(* Logix 5000 project; controller HP_SSC01 vendor 1 type 14 code 67 rev 17.7; software revision 17.01; part 12 of 15 *)
(* tags used below, declared in another part *)
   A_C1_0200 : ALIAS FOR S_C1_FaultSafety.0;
   A_C1_0201 : ALIAS FOR S_C1_FaultSafety.1;
   A_C1_0202 : ALIAS FOR S_C1_FaultSafety.2;
   A_C1_0203 : ALIAS FOR S_C1_FaultSafety.3;
   A_C1_0204 : ALIAS FOR S_C1_FaultSafety.4;
   A_C1_0206 : ALIAS FOR S_C1_FaultSafety.6;
   A_C1_0208 : ALIAS FOR S_C1_FaultSafety.8;
   A_C1_0209 : ALIAS FOR S_C1_FaultSafety.9;
   A_C1_0210 : ALIAS FOR S_C1_FaultSafety.10;
   A_C1_0211 : ALIAS FOR S_C1_FaultSafety.11;
   A_C1_0216 : ALIAS FOR S_C1_FaultSafety.16;
   A_C1_0217 : ALIAS FOR S_C1_FaultSafety.17;
   A_C1_0218 : ALIAS FOR S_C1_FaultSafety.18;
   A_C1_0219 : ALIAS FOR S_C1_FaultSafety.19;
   A_C1_0220 : ALIAS FOR S_C1_FaultSafety.20;
   A_C1_0221 : ALIAS FOR S_C1_FaultSafety.21;
   A_C1_0222 : ALIAS FOR S_C1_FaultSafety.22;
   A_C1_0223 : ALIAS FOR S_C1_FaultSafety.23;
   A_C1_0224 : ALIAS FOR S_C1_FaultSafety.24;
   A_C1_0230 : ALIAS FOR S_C1_FaultSafety.30;
   A_C1_0231 : ALIAS FOR S_C1_FaultSafety.31;
   A_C2_0200 : ALIAS FOR S_C2_FaultSafety.0;
   A_C2_0201 : ALIAS FOR S_C2_FaultSafety.1;
   A_C2_0210 : ALIAS FOR S_C2_FaultSafety.10;
   A_C2_0211 : ALIAS FOR S_C2_FaultSafety.11;
   A_C3_0200 : ALIAS FOR S_C3_FaultSafety.0;
   A_C3_0201 : ALIAS FOR S_C3_FaultSafety.1;
   A_C3_0210 : ALIAS FOR S_C3_FaultSafety.10;
   A_C3_0211 : ALIAS FOR S_C3_FaultSafety.11;
   A_S01_0103 : ALIAS FOR System_FaultSafeIO.3;
   A_S01_0104 : ALIAS FOR System_FaultSafeIO.4;
   A_S01_0105 : ALIAS FOR System_FaultSafeIO.5;
   A_S01_0116 : ALIAS FOR System_FaultSafeIO.16;
   A_S01_0117 : ALIAS FOR System_FaultSafeIO.17;
   A_S01_0118 : ALIAS FOR System_FaultSafeIO.18;
   A_S01_0119 : ALIAS FOR System_FaultSafeIO.19;
   A_S01_0120 : ALIAS FOR System_FaultSafeIO.20;
   A_S01_0122 : ALIAS FOR System_FaultSafeIO.22;
   A_S01_0123 : ALIAS FOR System_FaultSafeIO.23;
   A_S01_0124 : ALIAS FOR System_FaultSafeIO.24;
   A_S01_0201 : ALIAS FOR System_FaultSafety.1;
   A_S01_0204 : ALIAS FOR System_FaultSafety.4;
   A_S01_0206 : ALIAS FOR System_FaultSafety.6;
   A_S01_0208 : ALIAS FOR System_FaultSafety.8;
   A_S01_0209 : ALIAS FOR System_FaultSafety.9;
   A_S01_0210 : ALIAS FOR System_FaultSafety.10;
   A_S01_0211 : ALIAS FOR System_FaultSafety.11;
   A_S01_0212 : ALIAS FOR System_FaultSafety.12;
   A_S01_0213 : ALIAS FOR System_FaultSafety.13;
   A_S01_0216 : ALIAS FOR System_FaultSafety.16;
   C01_SafeMemory : Udt_Carsl_SafeData;
   ONS_STFault : DINT;
   Rail_Bypass1 : ALIAS FOR SSC01_Safe1:I.Pt06Data;
   Rail_Bypass2 : ALIAS FOR SSC01_Safe1:I.Pt07Data;
   RAIL_ENABLE_LH1 : ALIAS FOR SSC01_Safe1:I.Pt00Data;
   RAIL_ENABLE_LH2 : ALIAS FOR SSC01_Safe1:I.Pt01Data;
   RAIL_ENABLE_LH3 : ALIAS FOR SSC01_Safe1:I.Pt02Data;
   RAIL_ENABLE_RH1 : ALIAS FOR SSC01_Safe1:I.Pt03Data;
   RAIL_ENABLE_RH2 : ALIAS FOR SSC01_Safe1:I.Pt04Data;
   RAIL_ENABLE_RH3 : ALIAS FOR SSC01_Safe1:I.Pt05Data;
   RAIL_SHUNT_FDBK_LH1 : ALIAS FOR SSC01_Safe3:I.Pt00Data;
   RAIL_SHUNT_FDBK_LH2 : ALIAS FOR SSC01_Safe3:I.Pt01Data;
   RAIL_SHUNT_FDBK_LH3 : ALIAS FOR SSC01_Safe3:I.Pt02Data;
   Rail_Shunt_Fdbk_OK : BOOL;
   RAIL_SHUNT_FDBK_RH1 : ALIAS FOR SSC01_Safe3:I.Pt03Data;
   RAIL_SHUNT_FDBK_RH2 : ALIAS FOR SSC01_Safe3:I.Pt04Data;
   RAIL_SHUNT_FDBK_RH3 : ALIAS FOR SSC01_Safe3:I.Pt05Data;
   RAIL_SHUNT_LH1 : ALIAS FOR SSC01_Safe1:O.Pt00Data;
   RAIL_SHUNT_LH2 : ALIAS FOR SSC01_Safe1:O.Pt01Data;
   RAIL_SHUNT_LH3 : ALIAS FOR SSC01_Safe1:O.Pt02Data;
   RAIL_SHUNT_RH1 : ALIAS FOR SSC01_Safe1:O.Pt03Data;
   RAIL_SHUNT_RH2 : ALIAS FOR SSC01_Safe1:O.Pt04Data;
   RAIL_SHUNT_RH3 : ALIAS FOR SSC01_Safe1:O.Pt05Data;
   RCS_CMD_EvacToStation : BOOL;
   RCS_CMD_GoNearOnPath : BOOL;
   RCS_Cmd_Mismatch_TON : TIMER;
   RCS_CMD_RunInAuto : BOOL;
   RCS_Cmd_Unknown : BOOL;
   RCS_MasterClock : ALIAS FOR RCS_SafeMemory_S01.Master_Clock;
   RCS_MasterPositionMOD7000 : DINT;
   RCS_MasterPositionMOD7000X1000 : DINT;
   RCS_PwrDisc_RIN : REDUNDANT_INPUT;
   RCS_SafeMemory_S01 : Udt_RCS_SafeData;
   RCS_SyncMotionEnable : BOOL;
   S_C01_MStopOK : BOOL;
   S_C02_MStopOK : BOOL;
   S_C03_MStopOK : BOOL;
   S_C1_AtEvacSpeed : BOOL;
   S_C1_BrakeRelease : ALIAS FOR C1_Safe:O.Pt06Data;
   S_C1_BrakeReleaseSelected : BOOL;
   S_C1_BrakeTest : BOOL;
   S_C1_CircuitReset : BOOL;
   S_C1_DrawbridgeInputOK : BOOL;
   S_C1_DrawbridgeRIN : REDUNDANT_INPUT;
   S_C1_DumpValveRelease : ALIAS FOR C1_Safe:O.Pt05Data;
   S_C1_DumpValveReleaseSelected : BOOL;
   S_C1_EncoderBuffer : DINT[4];
   S_C1_EncoderChange : DINT;
   S_C1_EncoderCounter : DINT;
   S_C1_EncoderCounts : DINT;
   S_C1_EncoderPositionAtHome : DINT;
   S_C1_EncoderPositionAtHomeSet : BOOL;
   S_C1_EncoderPositionDegree : DINT;
   S_C1_EncoderRev : DINT;
   S_C1_EncoderRevX1000 : DINT;
   S_C1_EncoderTemp : DINT;
   S_C1_EncoderTemp2 : DINT;
   S_C1_EvacOk : BOOL;
   S_C1_ExecuteInputOK : BOOL;
   S_C1_FaultReset : BOOL;
   S_C1_FaultSafety : DINT;
   S_C1_FaultSafety_OK : BOOL;
   S_C1_FaultStandard_OK : BOOL;
   S_C1_FaultTimer : TIMER[8];
   S_C1_Homed : BOOL;
   S_C1_HomeInputStatus : BOOL;
   S_C1_HomeSafePE : ALIAS FOR C1_Safe:I.Pt04Data;
   S_C1_InEvacPosition : BOOL;
   S_C1_ModeLocal : BOOL;
   S_C1_ModeRemote : BOOL;
   S_C1_MotorActualPositionX1000 : DINT;
   S_C1_MotorAverageVelocityX1000 : DINT;
   S_C1_MotorToEncoderError : DINT;
   S_C1_MStop : EMERGENCY_STOP;
   S_C1_MSTOP_InputOK : BOOL;
   S_C1_OffPath : BOOL;
   S_C1_OnPath : BOOL;
   S_C1_ONS_Fault : BOOL;
   S_C1_OutputEnable : BOOL;
   S_C1_PressureOK : ALIAS FOR C1_Safe:I.Pt05Data;
   S_C1_RemoteBrakeAndHomeSequence : DINT;
   S_C1_ReverseMotionDebounce : TIMER;
   S_C1_SAFE_OFF_FDBK1 : ALIAS FOR C1_Safe:I.Pt01Data;
   S_C1_SAFE_OFF_FDBK2 : ALIAS FOR C1_Safe:I.Pt00Data;
   S_C1_SafeOff_ROUT : REDUNDANT_OUTPUT;
   S_C1_SafeOffInputOK : BOOL;
   S_C1_SetEncoderHomePosition : BOOL;
   S_C1_Stop0 : BOOL;
   S_C1_Stop0_OK : BOOL;
   S_C1_Stop1 : BOOL;
   S_C1_Stop1_OK : BOOL;
   S_C2_EvacOK : BOOL;
   S_C2_ModeLocal : BOOL;
   S_C2_ModeRemote : BOOL;
   S_C2_OffPath : BOOL;
   S_C2_OnPath : BOOL;
   S_C2_Stop0 : BOOL;
   S_C2_Stop0_OK : BOOL;
   S_C2_Stop1 : BOOL;
   S_C2_Stop1_OK : BOOL;
   S_C3_EvacOK : BOOL;
   S_C3_ModeLocal : BOOL;
   S_C3_ModeRemote : BOOL;
   S_C3_OffPath : BOOL;
   S_C3_OnPath : BOOL;
   S_C3_Stop0 : BOOL;
   S_C3_Stop0_OK : BOOL;
   S_C3_Stop1 : BOOL;
   S_C3_Stop1_OK : BOOL;
   S_DeviceNet_OK : BOOL;
   S_EncoderRollover : DINT;
   S_EvacToStationTON : TIMER;
   S_FaultReset : BOOL;
   S_RCS_EvacSpeedStart_TON : TIMER;
   S_RCS_MasterPositionDegrees : DINT;
   S_S01_Mode_Remote : BOOL;
   S_S01_NearOnPath : BOOL;
   S_S01_OnPath : BOOL;
   S_S01_Ready : BOOL;
   S_System_FaultStandard : DINT;
   SSC_Auto_Decel1 : BOOL;
   SSC_Mode_Local_LT : ALIAS FOR SSC01_Safe3:O.Pt00Data;
   SSC_Mode_Remote_LT : ALIAS FOR SSC01_Safe3:O.Pt02Data;
   SSC_NoStopFault : BOOL;
   SSC_Rail_BypassOK : BOOL;
   SSC_Rail_InputsOK : BOOL;
   SSC_RailShuntOK : BOOL;
   SSC_Ready_LT : ALIAS FOR SSC01_Safe3:O.Pt01Data;
   SSC_SafeFlt_OK : BOOL;
   SSC_SafetyIO_OK : BOOL;
   SSC_StdFlt_OK : BOOL;
   SSC_Stop0_OK : BOOL;
   SSC_Stop1_OK : BOOL;
   ST_NoScan_Comment : BOOL;
   STS_Rail_Bypass_InputOK : BOOL;
   STS_RCS_PwrDisc_InputOK : BOOL;
   STS_Status_OK : BOOL;
   System_FaultSafeIO : DINT;
   System_FaultSafety : DINT;
   Tmr_Rail_Shunt : TIMER[7];
(* Safe_SSC, continued *)

ROUTINE ST10_PositionHandling   (* ladder *)
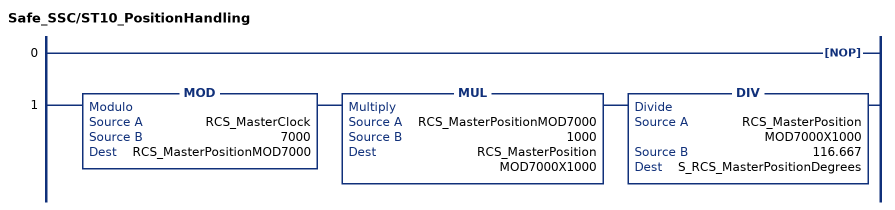
   0: NOP();
   1: MOD(RCS_MasterClock,7000,RCS_MasterPositionMOD7000)MUL(RCS_MasterPositionMOD7000,1000,RCS_MasterPositionMOD7000X1000)DIV(RCS_MasterPositionMOD7000X1000,116.667,S_RCS_MasterPositionDegrees);
END_ROUTINE

ROUTINE ST21_RailShunt   (* ladder *)
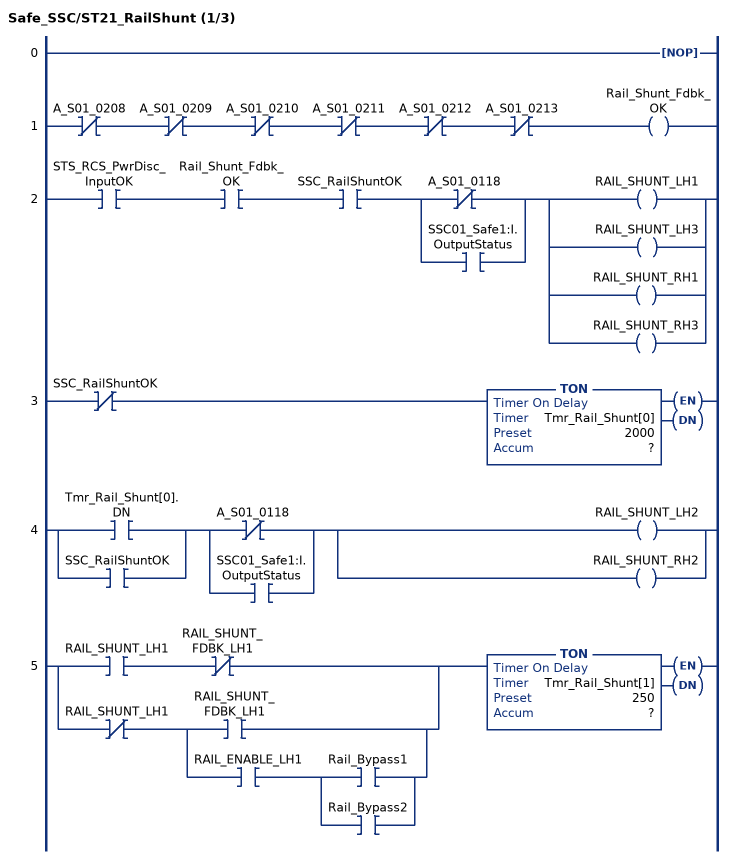
   0: NOP();
   1: XIO(A_S01_0208)XIO(A_S01_0209)XIO(A_S01_0210)XIO(A_S01_0211)XIO(A_S01_0212)XIO(A_S01_0213)OTE(Rail_Shunt_Fdbk_OK);
   2: XIC(STS_RCS_PwrDisc_InputOK)XIC(Rail_Shunt_Fdbk_OK)XIC(SSC_RailShuntOK)[XIO(A_S01_0118) ,XIC(SSC01_Safe1:I.OutputStatus) ][OTE(RAIL_SHUNT_LH1) ,OTE(RAIL_SHUNT_LH3) ,OTE(RAIL_SHUNT_RH1) ,OTE(RAIL_SHUNT_RH3) ];
   3: XIO(SSC_RailShuntOK)TON(Tmr_Rail_Shunt[0],?,?);
   4: [XIC(Tmr_Rail_Shunt[0].DN) ,XIC(SSC_RailShuntOK) ][XIO(A_S01_0118) ,XIC(SSC01_Safe1:I.OutputStatus) ][OTE(RAIL_SHUNT_LH2) ,OTE(RAIL_SHUNT_RH2) ];
   5: [XIC(RAIL_SHUNT_LH1) XIO(RAIL_SHUNT_FDBK_LH1) ,XIO(RAIL_SHUNT_LH1) [XIC(RAIL_SHUNT_FDBK_LH1) ,XIC(RAIL_ENABLE_LH1) [XIC(Rail_Bypass1) ,XIC(Rail_Bypass2) ] ] ]TON(Tmr_Rail_Shunt[1],?,?);
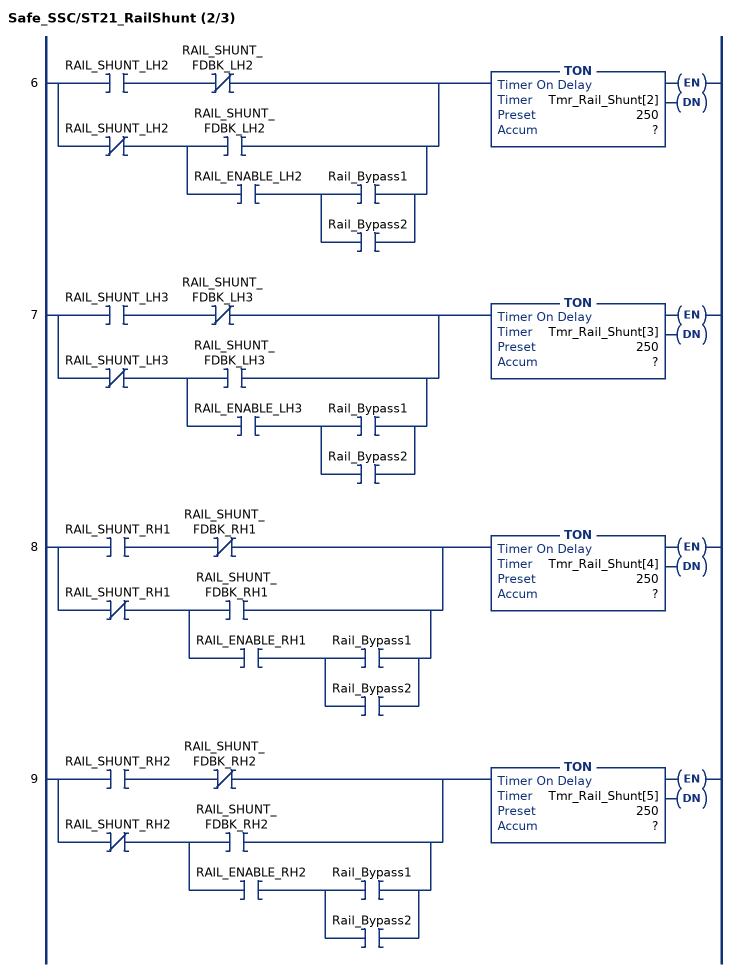
   6: [XIC(RAIL_SHUNT_LH2) XIO(RAIL_SHUNT_FDBK_LH2) ,XIO(RAIL_SHUNT_LH2) [XIC(RAIL_SHUNT_FDBK_LH2) ,XIC(RAIL_ENABLE_LH2) [XIC(Rail_Bypass1) ,XIC(Rail_Bypass2) ] ] ]TON(Tmr_Rail_Shunt[2],?,?);
   7: [XIC(RAIL_SHUNT_LH3) XIO(RAIL_SHUNT_FDBK_LH3) ,XIO(RAIL_SHUNT_LH3) [XIC(RAIL_SHUNT_FDBK_LH3) ,XIC(RAIL_ENABLE_LH3) [XIC(Rail_Bypass1) ,XIC(Rail_Bypass2) ] ] ]TON(Tmr_Rail_Shunt[3],?,?);
   8: [XIC(RAIL_SHUNT_RH1) XIO(RAIL_SHUNT_FDBK_RH1) ,XIO(RAIL_SHUNT_RH1) [XIC(RAIL_SHUNT_FDBK_RH1) ,XIC(RAIL_ENABLE_RH1) [XIC(Rail_Bypass1) ,XIC(Rail_Bypass2) ] ] ]TON(Tmr_Rail_Shunt[4],?,?);
   9: [XIC(RAIL_SHUNT_RH2) XIO(RAIL_SHUNT_FDBK_RH2) ,XIO(RAIL_SHUNT_RH2) [XIC(RAIL_SHUNT_FDBK_RH2) ,XIC(RAIL_ENABLE_RH2) [XIC(Rail_Bypass1) ,XIC(Rail_Bypass2) ] ] ]TON(Tmr_Rail_Shunt[5],?,?);
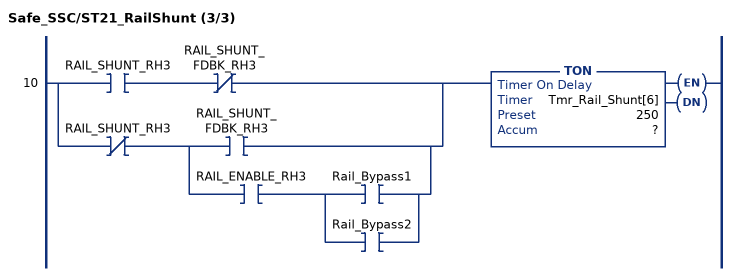
   10: [XIC(RAIL_SHUNT_RH3) XIO(RAIL_SHUNT_FDBK_RH3) ,XIO(RAIL_SHUNT_RH3) [XIC(RAIL_SHUNT_FDBK_RH3) ,XIC(RAIL_ENABLE_RH3) [XIC(Rail_Bypass1) ,XIC(Rail_Bypass2) ] ] ]TON(Tmr_Rail_Shunt[6],?,?);
END_ROUTINE

ROUTINE ST23_GenOutputs   (* ladder *)
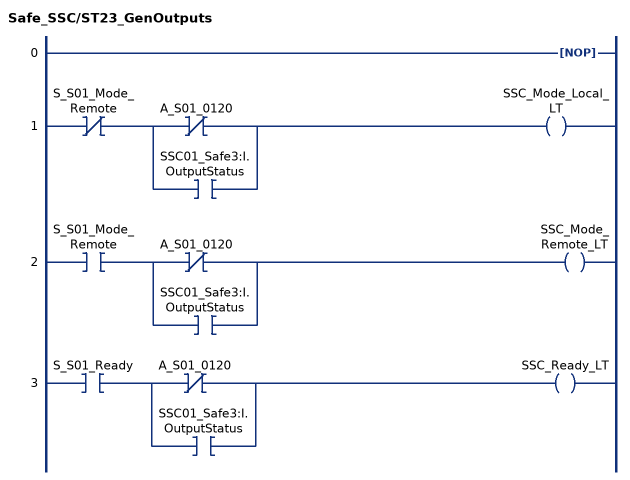
   0: NOP();
   1: XIO(S_S01_Mode_Remote)[XIO(A_S01_0120) ,XIC(SSC01_Safe3:I.OutputStatus) ]OTE(SSC_Mode_Local_LT);
   2: XIC(S_S01_Mode_Remote)[XIO(A_S01_0120) ,XIC(SSC01_Safe3:I.OutputStatus) ]OTE(SSC_Mode_Remote_LT);
   3: XIC(S_S01_Ready)[XIO(A_S01_0120) ,XIC(SSC01_Safe3:I.OutputStatus) ]OTE(SSC_Ready_LT);
END_ROUTINE

ROUTINE ST90_Faults   (* ladder *)
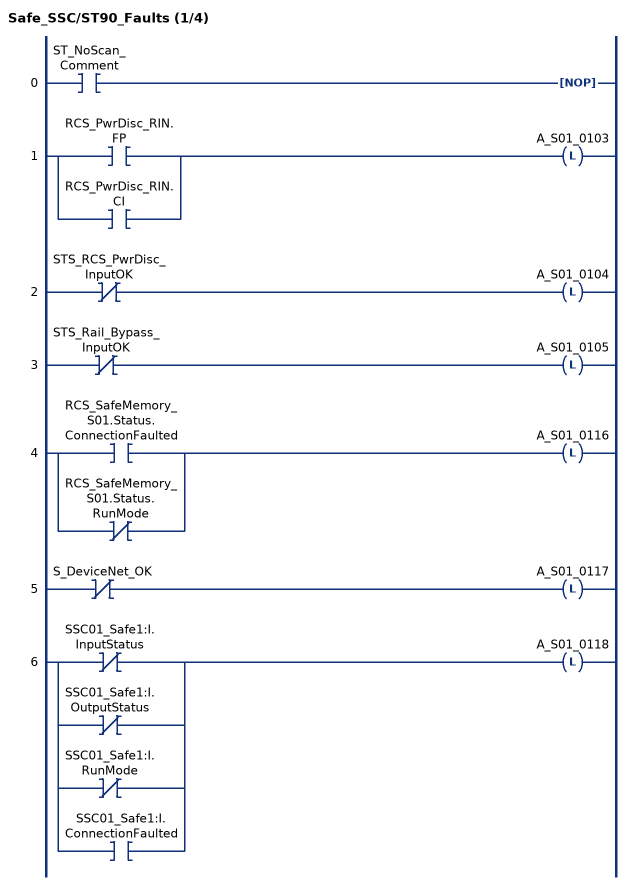
   0: XIC(ST_NoScan_Comment)NOP();
   1: [XIC(RCS_PwrDisc_RIN.FP) ,XIC(RCS_PwrDisc_RIN.CI) ]OTL(A_S01_0103);
   2: XIO(STS_RCS_PwrDisc_InputOK)OTL(A_S01_0104);
   3: XIO(STS_Rail_Bypass_InputOK)OTL(A_S01_0105);
   4: [XIC(RCS_SafeMemory_S01.Status.ConnectionFaulted) ,XIO(RCS_SafeMemory_S01.Status.RunMode) ]OTL(A_S01_0116);
   5: XIO(S_DeviceNet_OK)OTL(A_S01_0117);
   6: [XIO(SSC01_Safe1:I.InputStatus) ,XIO(SSC01_Safe1:I.OutputStatus) ,XIO(SSC01_Safe1:I.RunMode) ,XIC(SSC01_Safe1:I.ConnectionFaulted) ]OTL(A_S01_0118);
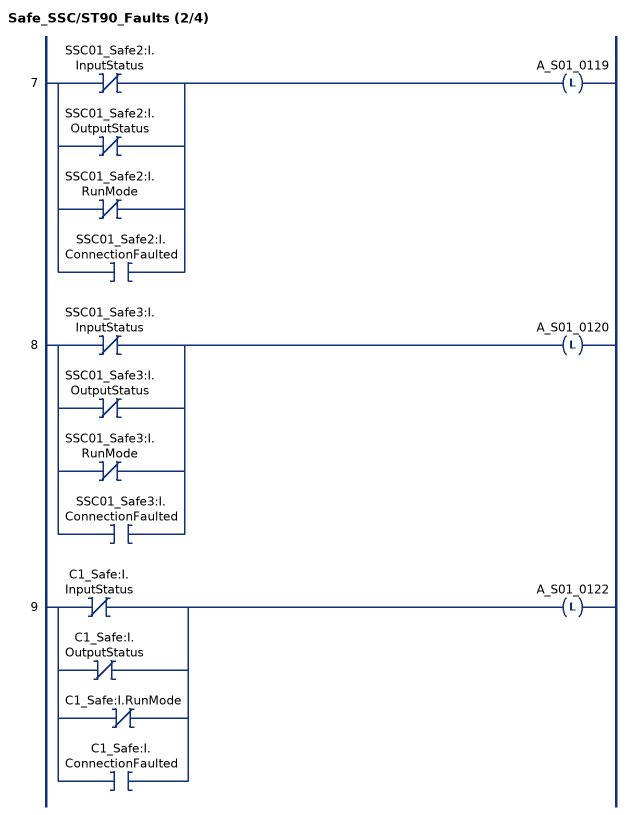
   7: [XIO(SSC01_Safe2:I.InputStatus) ,XIO(SSC01_Safe2:I.OutputStatus) ,XIO(SSC01_Safe2:I.RunMode) ,XIC(SSC01_Safe2:I.ConnectionFaulted) ]OTL(A_S01_0119);
   8: [XIO(SSC01_Safe3:I.InputStatus) ,XIO(SSC01_Safe3:I.OutputStatus) ,XIO(SSC01_Safe3:I.RunMode) ,XIC(SSC01_Safe3:I.ConnectionFaulted) ]OTL(A_S01_0120);
   9: [XIO(C1_Safe:I.InputStatus) ,XIO(C1_Safe:I.OutputStatus) ,XIO(C1_Safe:I.RunMode) ,XIC(C1_Safe:I.ConnectionFaulted) ]OTL(A_S01_0122);
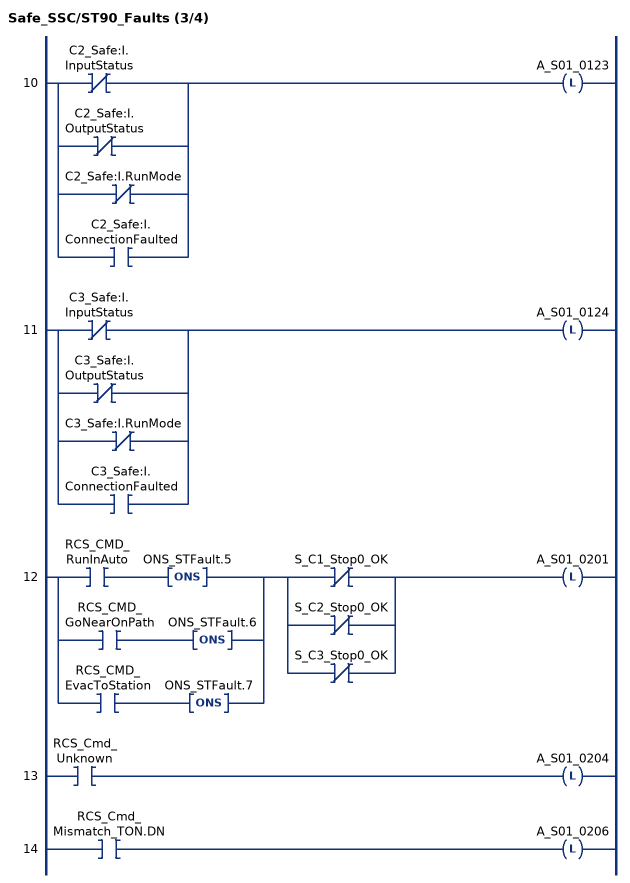
   10: [XIO(C2_Safe:I.InputStatus) ,XIO(C2_Safe:I.OutputStatus) ,XIO(C2_Safe:I.RunMode) ,XIC(C2_Safe:I.ConnectionFaulted) ]OTL(A_S01_0123);
   11: [XIO(C3_Safe:I.InputStatus) ,XIO(C3_Safe:I.OutputStatus) ,XIO(C3_Safe:I.RunMode) ,XIC(C3_Safe:I.ConnectionFaulted) ]OTL(A_S01_0124);
   12: [XIC(RCS_CMD_RunInAuto) ONS(ONS_STFault.5) ,XIC(RCS_CMD_GoNearOnPath) ONS(ONS_STFault.6) ,XIC(RCS_CMD_EvacToStation) ONS(ONS_STFault.7) ][XIO(S_C1_Stop0_OK) ,XIO(S_C2_Stop0_OK) ,XIO(S_C3_Stop0_OK) ]OTL(A_S01_0201);
   13: XIC(RCS_Cmd_Unknown)OTL(A_S01_0204);
   14: XIC(RCS_Cmd_Mismatch_TON.DN)OTL(A_S01_0206);
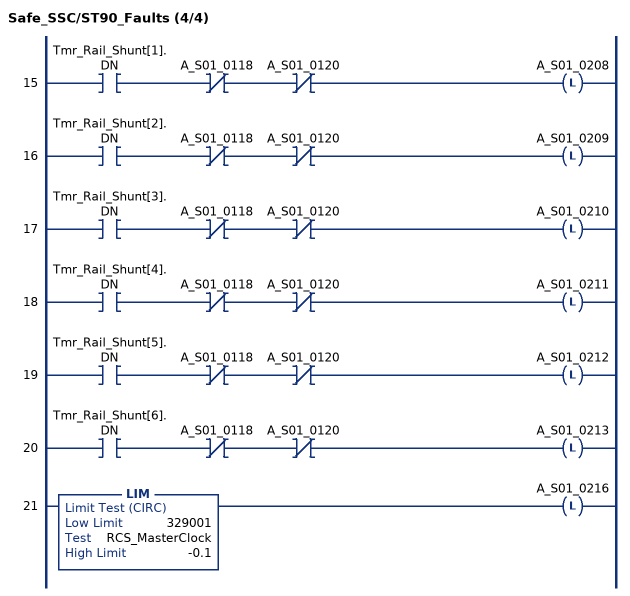
   15: XIC(Tmr_Rail_Shunt[1].DN)XIO(A_S01_0118)XIO(A_S01_0120)OTL(A_S01_0208);
   16: XIC(Tmr_Rail_Shunt[2].DN)XIO(A_S01_0118)XIO(A_S01_0120)OTL(A_S01_0209);
   17: XIC(Tmr_Rail_Shunt[3].DN)XIO(A_S01_0118)XIO(A_S01_0120)OTL(A_S01_0210);
   18: XIC(Tmr_Rail_Shunt[4].DN)XIO(A_S01_0118)XIO(A_S01_0120)OTL(A_S01_0211);
   19: XIC(Tmr_Rail_Shunt[5].DN)XIO(A_S01_0118)XIO(A_S01_0120)OTL(A_S01_0212);
   20: XIC(Tmr_Rail_Shunt[6].DN)XIO(A_S01_0118)XIO(A_S01_0120)OTL(A_S01_0213);
   21: LIM(329001,RCS_MasterClock,-0.1)OTL(A_S01_0216);
END_ROUTINE

ROUTINE ST91_FaultList   (* ladder *)
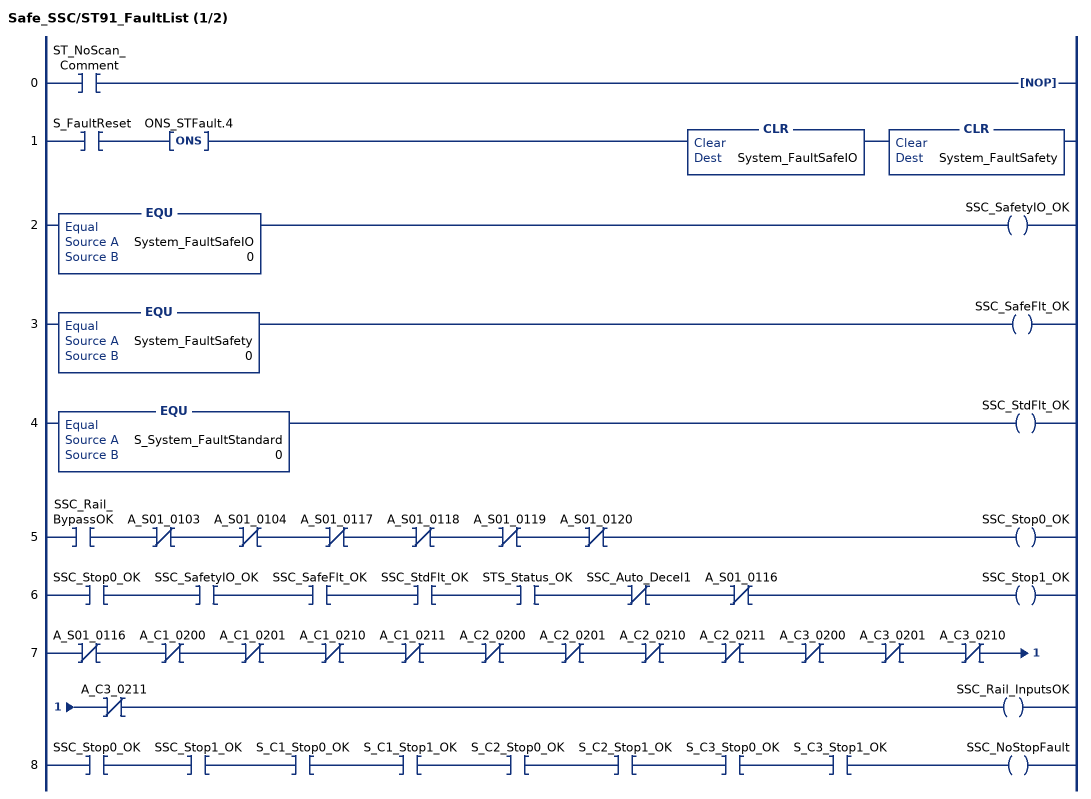
   0: XIC(ST_NoScan_Comment)NOP();
   1: XIC(S_FaultReset)ONS(ONS_STFault.4)CLR(System_FaultSafeIO)CLR(System_FaultSafety);
   2: EQU(System_FaultSafeIO,0)OTE(SSC_SafetyIO_OK);
   3: EQU(System_FaultSafety,0)OTE(SSC_SafeFlt_OK);
   4: EQU(S_System_FaultStandard,0)OTE(SSC_StdFlt_OK);
   5: XIC(SSC_Rail_BypassOK)XIO(A_S01_0103)XIO(A_S01_0104)XIO(A_S01_0117)XIO(A_S01_0118)XIO(A_S01_0119)XIO(A_S01_0120)OTE(SSC_Stop0_OK);
   6: XIC(SSC_Stop0_OK)XIC(SSC_SafetyIO_OK)XIC(SSC_SafeFlt_OK)XIC(SSC_StdFlt_OK)XIC(STS_Status_OK)XIO(SSC_Auto_Decel1)XIO(A_S01_0116)OTE(SSC_Stop1_OK);
   7: XIO(A_S01_0116)XIO(A_C1_0200)XIO(A_C1_0201)XIO(A_C1_0210)XIO(A_C1_0211)XIO(A_C2_0200)XIO(A_C2_0201)XIO(A_C2_0210)XIO(A_C2_0211)XIO(A_C3_0200)XIO(A_C3_0201)XIO(A_C3_0210)XIO(A_C3_0211)OTE(SSC_Rail_InputsOK);
   8: XIC(SSC_Stop0_OK)XIC(SSC_Stop1_OK)XIC(S_C1_Stop0_OK)XIC(S_C1_Stop1_OK)XIC(S_C2_Stop0_OK)XIC(S_C2_Stop1_OK)XIC(S_C3_Stop0_OK)XIC(S_C3_Stop1_OK)OTE(SSC_NoStopFault);
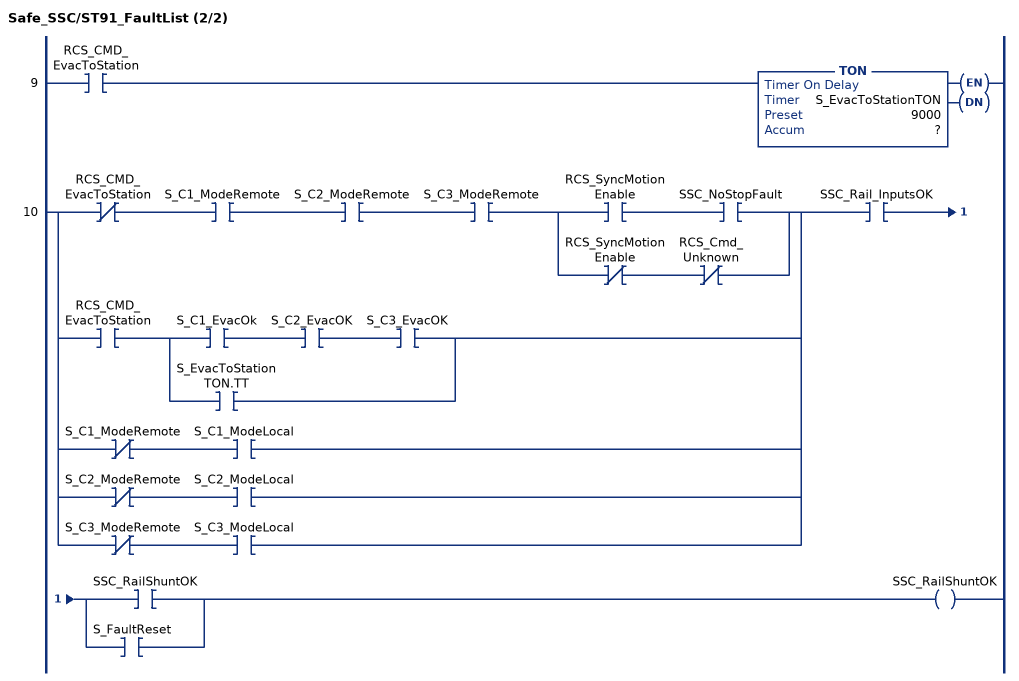
   9: XIC(RCS_CMD_EvacToStation)TON(S_EvacToStationTON,?,?);
   10: [XIO(RCS_CMD_EvacToStation) XIC(S_C1_ModeRemote) XIC(S_C2_ModeRemote) XIC(S_C3_ModeRemote) [XIC(RCS_SyncMotionEnable) XIC(SSC_NoStopFault) ,XIO(RCS_SyncMotionEnable) XIO(RCS_Cmd_Unknown) ] ,XIC(RCS_CMD_EvacToStation) [XIC(S_C1_EvacOk) XIC(S_C2_EvacOK) XIC(S_C3_EvacOK) ,XIC(S_EvacToStationTON.TT) ] ,XIO(S_C1_ModeRemote) XIC(S_C1_ModeLocal) ,XIO(S_C2_ModeRemote) XIC(S_C2_ModeLocal) ,XIO(S_C3_ModeRemote) XIC(S_C3_ModeLocal) ]XIC(SSC_Rail_InputsOK)[XIC(SSC_RailShuntOK) ,XIC(S_FaultReset) ]OTE(SSC_RailShuntOK);
END_ROUTINE

ROUTINE ST99_CommToRCS   (* ladder *)
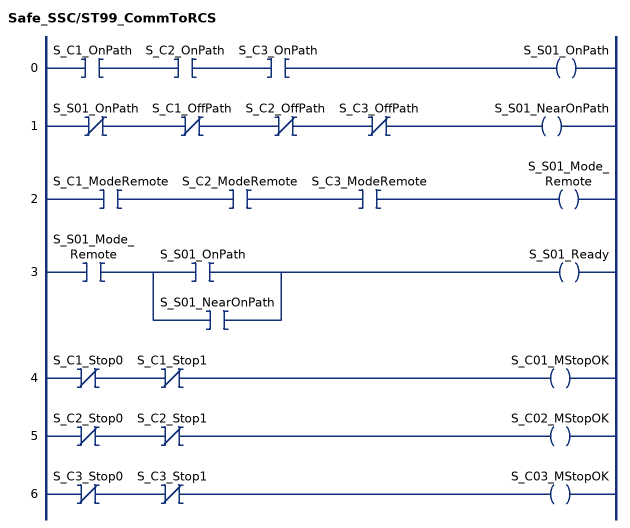
   0: XIC(S_C1_OnPath)XIC(S_C2_OnPath)XIC(S_C3_OnPath)OTE(S_S01_OnPath);
   1: XIO(S_S01_OnPath)XIO(S_C1_OffPath)XIO(S_C2_OffPath)XIO(S_C3_OffPath)OTE(S_S01_NearOnPath);
   2: XIC(S_C1_ModeRemote)XIC(S_C2_ModeRemote)XIC(S_C3_ModeRemote)OTE(S_S01_Mode_Remote);
   3: XIC(S_S01_Mode_Remote)[XIC(S_S01_OnPath) ,XIC(S_S01_NearOnPath) ]OTE(S_S01_Ready);
   4: XIO(S_C1_Stop0)XIO(S_C1_Stop1)OTE(S_C01_MStopOK);
   5: XIO(S_C2_Stop0)XIO(S_C2_Stop1)OTE(S_C02_MStopOK);
   6: XIO(S_C3_Stop0)XIO(S_C3_Stop1)OTE(S_C03_MStopOK);
END_ROUTINE
END_PROGRAM

PROGRAM SafeCarousel1   (* main routine SC100_Main *)

ROUTINE SC100_Main   (* ladder *)
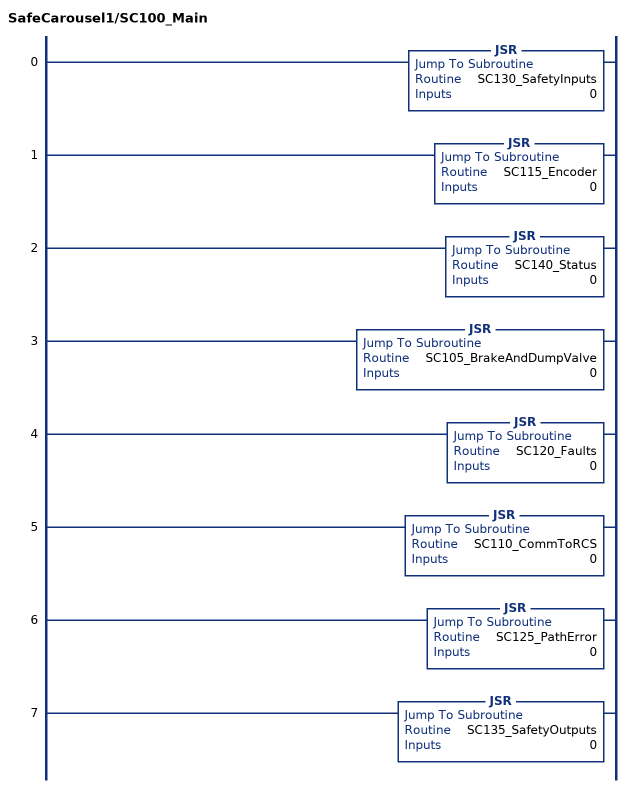
   0: JSR(SC130_SafetyInputs,0);
   1: JSR(SC115_Encoder,0);
   2: JSR(SC140_Status,0);
   3: JSR(SC105_BrakeAndDumpValve,0);
   4: JSR(SC120_Faults,0);
   5: JSR(SC110_CommToRCS,0);
   6: JSR(SC125_PathError,0);
   7: JSR(SC135_SafetyOutputs,0);
END_ROUTINE

ROUTINE SC105_BrakeAndDumpValve   (* ladder *)
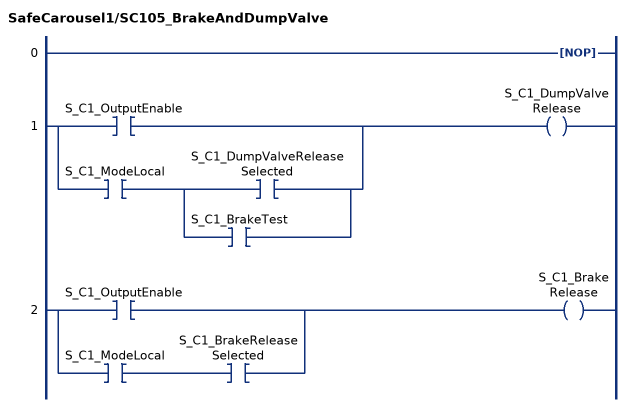
   0: NOP();
   1: [XIC(S_C1_OutputEnable) ,XIC(S_C1_ModeLocal) [XIC(S_C1_DumpValveReleaseSelected) ,XIC(S_C1_BrakeTest) ] ]OTE(S_C1_DumpValveRelease);
   2: [XIC(S_C1_OutputEnable) ,XIC(S_C1_ModeLocal) XIC(S_C1_BrakeReleaseSelected) ]OTE(S_C1_BrakeRelease);
END_ROUTINE

ROUTINE SC110_CommToRCS   (* ladder *)
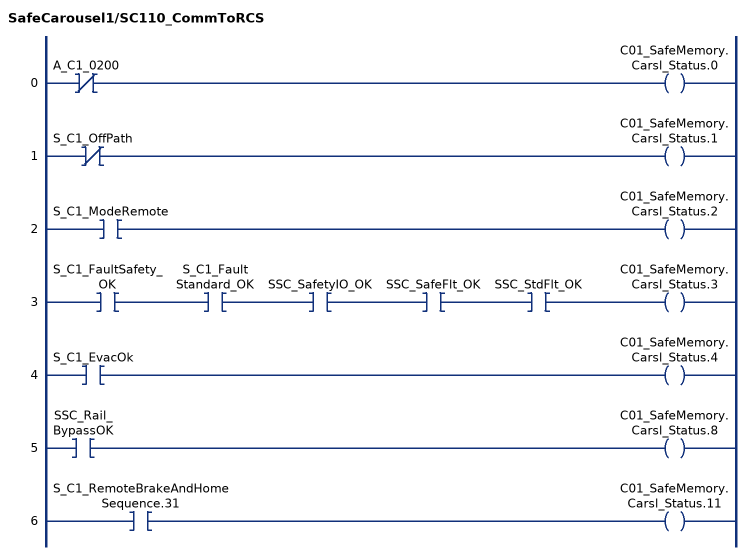
   0: XIO(A_C1_0200)OTE(C01_SafeMemory.Carsl_Status.0);
   1: XIO(S_C1_OffPath)OTE(C01_SafeMemory.Carsl_Status.1);
   2: XIC(S_C1_ModeRemote)OTE(C01_SafeMemory.Carsl_Status.2);
   3: XIC(S_C1_FaultSafety_OK)XIC(S_C1_FaultStandard_OK)XIC(SSC_SafetyIO_OK)XIC(SSC_SafeFlt_OK)XIC(SSC_StdFlt_OK)OTE(C01_SafeMemory.Carsl_Status.3);
   4: XIC(S_C1_EvacOk)OTE(C01_SafeMemory.Carsl_Status.4);
   5: XIC(SSC_Rail_BypassOK)OTE(C01_SafeMemory.Carsl_Status.8);
   6: XIC(S_C1_RemoteBrakeAndHomeSequence.31)OTE(C01_SafeMemory.Carsl_Status.11);
END_ROUTINE

ROUTINE SC115_Encoder   (* ladder *)
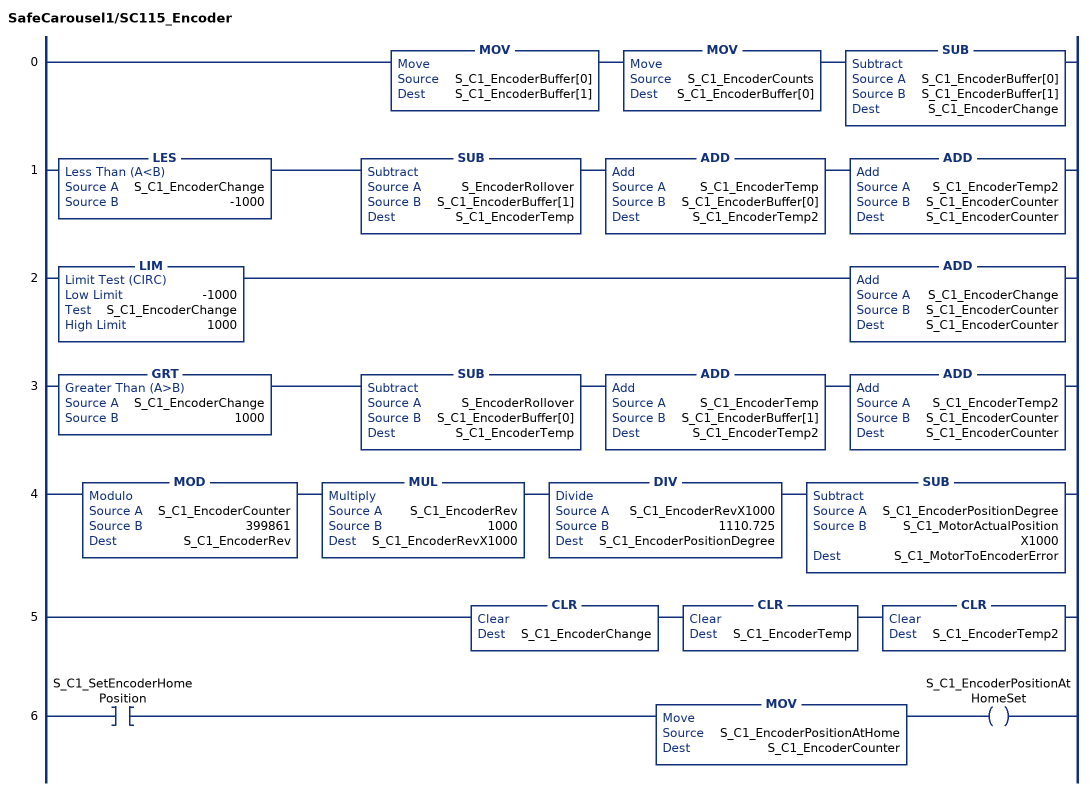
   0: MOV(S_C1_EncoderBuffer[0],S_C1_EncoderBuffer[1])MOV(S_C1_EncoderCounts,S_C1_EncoderBuffer[0])SUB(S_C1_EncoderBuffer[0],S_C1_EncoderBuffer[1],S_C1_EncoderChange);
   1: LES(S_C1_EncoderChange,-1000)SUB(S_EncoderRollover,S_C1_EncoderBuffer[1],S_C1_EncoderTemp)ADD(S_C1_EncoderTemp,S_C1_EncoderBuffer[0],S_C1_EncoderTemp2)ADD(S_C1_EncoderTemp2,S_C1_EncoderCounter,S_C1_EncoderCounter);
   2: LIM(-1000,S_C1_EncoderChange,1000)ADD(S_C1_EncoderChange,S_C1_EncoderCounter,S_C1_EncoderCounter);
   3: GRT(S_C1_EncoderChange,1000)SUB(S_EncoderRollover,S_C1_EncoderBuffer[0],S_C1_EncoderTemp)ADD(S_C1_EncoderTemp,S_C1_EncoderBuffer[1],S_C1_EncoderTemp2)ADD(S_C1_EncoderTemp2,S_C1_EncoderCounter,S_C1_EncoderCounter);
   4: MOD(S_C1_EncoderCounter,399861,S_C1_EncoderRev)MUL(S_C1_EncoderRev,1000,S_C1_EncoderRevX1000)DIV(S_C1_EncoderRevX1000,1110.725,S_C1_EncoderPositionDegree)SUB(S_C1_EncoderPositionDegree,S_C1_MotorActualPositionX1000,S_C1_MotorToEncoderError);
   5: CLR(S_C1_EncoderChange)CLR(S_C1_EncoderTemp)CLR(S_C1_EncoderTemp2);
   6: XIC(S_C1_SetEncoderHomePosition)MOV(S_C1_EncoderPositionAtHome,S_C1_EncoderCounter)OTE(S_C1_EncoderPositionAtHomeSet);
END_ROUTINE

ROUTINE SC120_Faults   (* ladder *)
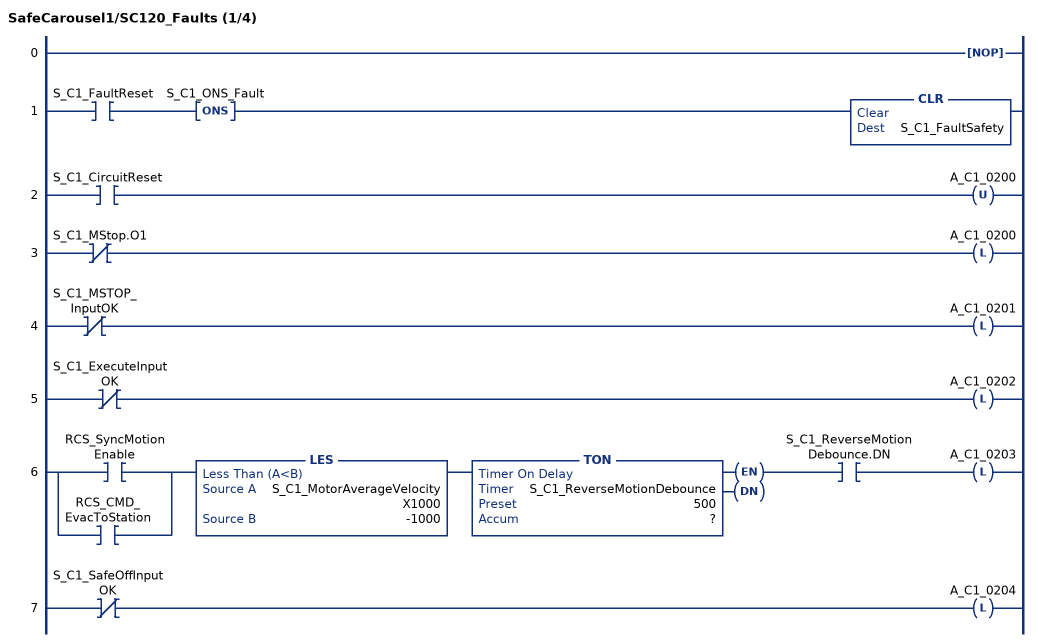
   0: NOP();
   1: XIC(S_C1_FaultReset)ONS(S_C1_ONS_Fault)CLR(S_C1_FaultSafety);
   2: XIC(S_C1_CircuitReset)OTU(A_C1_0200);
   3: XIO(S_C1_MStop.O1)OTL(A_C1_0200);
   4: XIO(S_C1_MSTOP_InputOK)OTL(A_C1_0201);
   5: XIO(S_C1_ExecuteInputOK)OTL(A_C1_0202);
   6: [XIC(RCS_SyncMotionEnable) ,XIC(RCS_CMD_EvacToStation) ]LES(S_C1_MotorAverageVelocityX1000,-1000)TON(S_C1_ReverseMotionDebounce,?,?)XIC(S_C1_ReverseMotionDebounce.DN)OTL(A_C1_0203);
   7: XIO(S_C1_SafeOffInputOK)OTL(A_C1_0204);
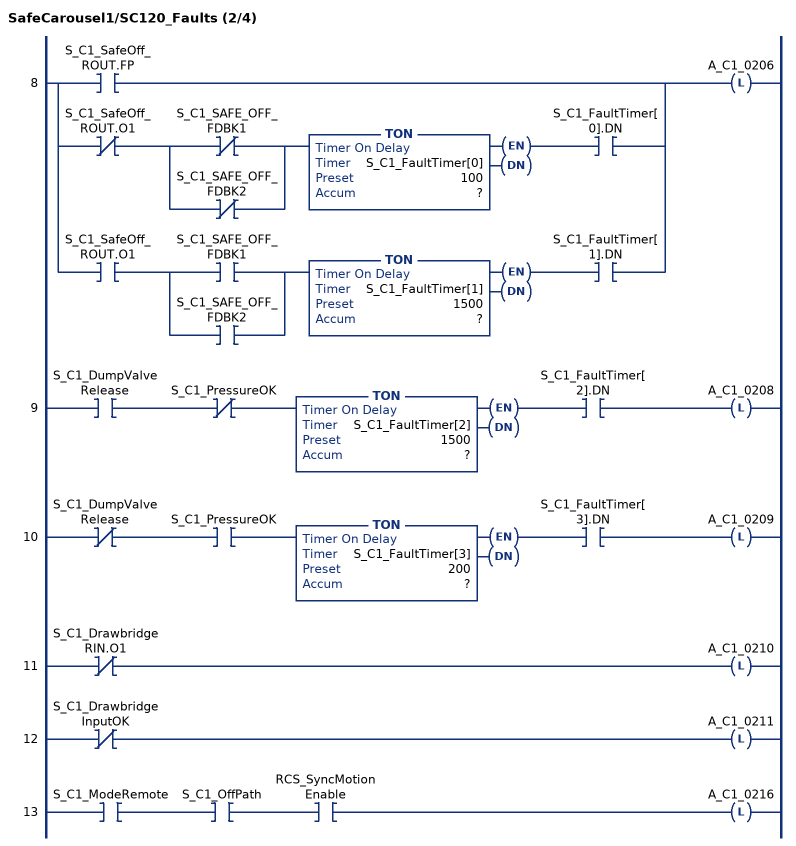
   8: [XIC(S_C1_SafeOff_ROUT.FP) ,XIO(S_C1_SafeOff_ROUT.O1) [XIO(S_C1_SAFE_OFF_FDBK1) ,XIO(S_C1_SAFE_OFF_FDBK2) ] TON(S_C1_FaultTimer[0],?,?) XIC(S_C1_FaultTimer[0].DN) ,XIC(S_C1_SafeOff_ROUT.O1) [XIC(S_C1_SAFE_OFF_FDBK1) ,XIC(S_C1_SAFE_OFF_FDBK2) ] TON(S_C1_FaultTimer[1],?,?) XIC(S_C1_FaultTimer[1].DN) ]OTL(A_C1_0206);
   9: XIC(S_C1_DumpValveRelease)XIO(S_C1_PressureOK)TON(S_C1_FaultTimer[2],?,?)XIC(S_C1_FaultTimer[2].DN)OTL(A_C1_0208);
   10: XIO(S_C1_DumpValveRelease)XIC(S_C1_PressureOK)TON(S_C1_FaultTimer[3],?,?)XIC(S_C1_FaultTimer[3].DN)OTL(A_C1_0209);
   11: XIO(S_C1_DrawbridgeRIN.O1)OTL(A_C1_0210);
   12: XIO(S_C1_DrawbridgeInputOK)OTL(A_C1_0211);
   13: XIC(S_C1_ModeRemote)XIC(S_C1_OffPath)XIC(RCS_SyncMotionEnable)OTL(A_C1_0216);
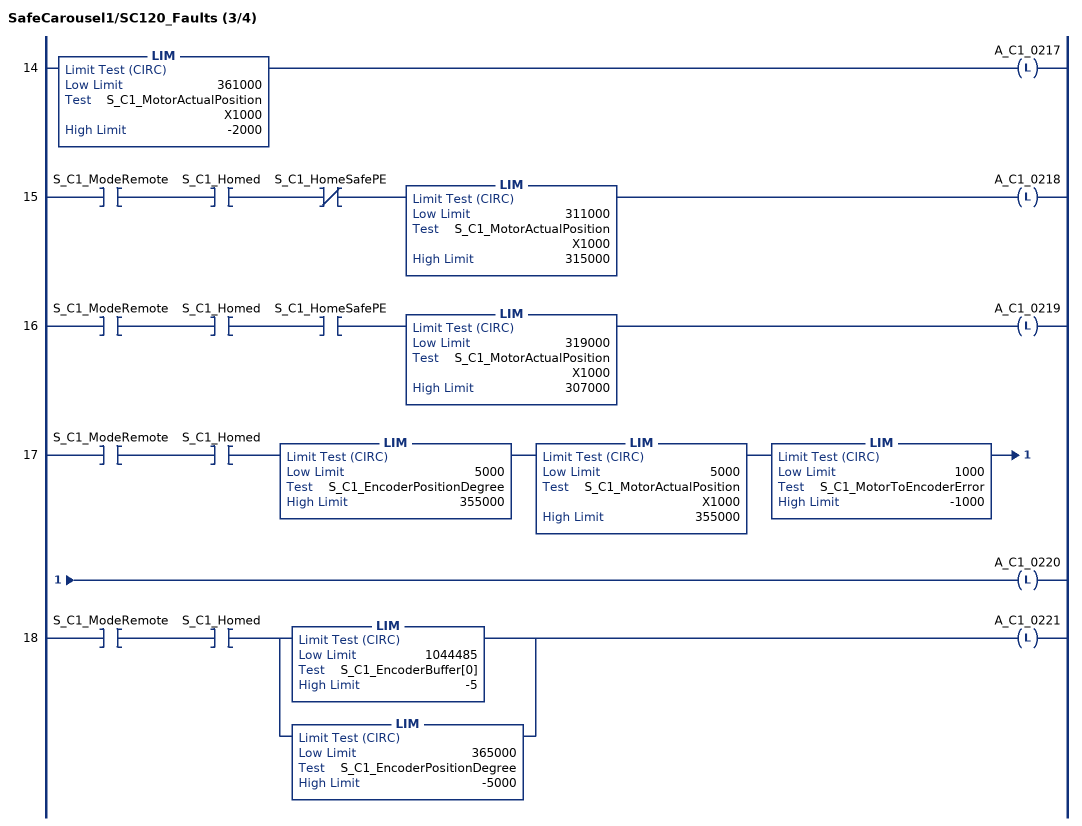
   14: LIM(361000,S_C1_MotorActualPositionX1000,-2000)OTL(A_C1_0217);
   15: XIC(S_C1_ModeRemote)XIC(S_C1_Homed)XIO(S_C1_HomeSafePE)LIM(311000,S_C1_MotorActualPositionX1000,315000)OTL(A_C1_0218);
   16: XIC(S_C1_ModeRemote)XIC(S_C1_Homed)XIC(S_C1_HomeSafePE)LIM(319000,S_C1_MotorActualPositionX1000,307000)OTL(A_C1_0219);
   17: XIC(S_C1_ModeRemote)XIC(S_C1_Homed)LIM(5000,S_C1_EncoderPositionDegree,355000)LIM(5000,S_C1_MotorActualPositionX1000,355000)LIM(1000,S_C1_MotorToEncoderError,-1000)OTL(A_C1_0220);
   18: XIC(S_C1_ModeRemote)XIC(S_C1_Homed)[LIM(1044485,S_C1_EncoderBuffer[0],-5) ,LIM(365000,S_C1_EncoderPositionDegree,-5000) ]OTL(A_C1_0221);
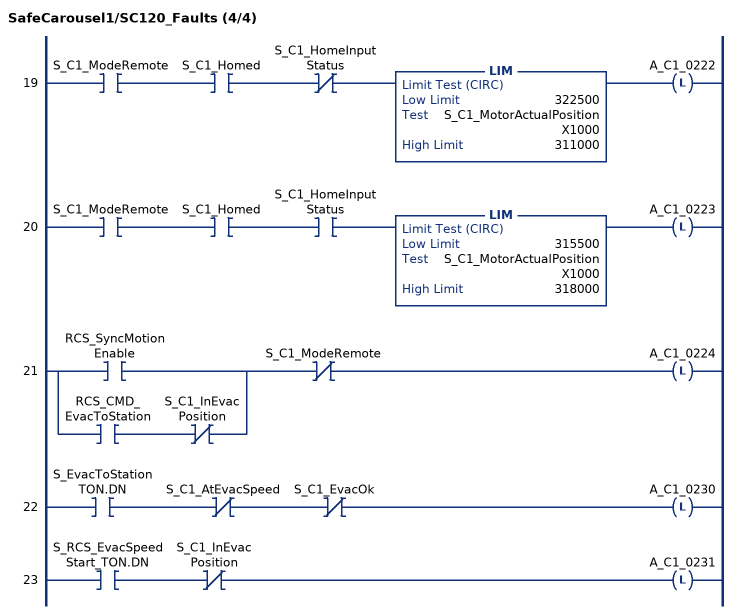
   19: XIC(S_C1_ModeRemote)XIC(S_C1_Homed)XIO(S_C1_HomeInputStatus)LIM(322500,S_C1_MotorActualPositionX1000,311000)OTL(A_C1_0222);
   20: XIC(S_C1_ModeRemote)XIC(S_C1_Homed)XIC(S_C1_HomeInputStatus)LIM(315500,S_C1_MotorActualPositionX1000,318000)OTL(A_C1_0223);
   21: [XIC(RCS_SyncMotionEnable) ,XIC(RCS_CMD_EvacToStation) XIO(S_C1_InEvacPosition) ]XIO(S_C1_ModeRemote)OTL(A_C1_0224);
   22: XIC(S_EvacToStationTON.DN)XIO(S_C1_AtEvacSpeed)XIO(S_C1_EvacOk)OTL(A_C1_0230);
   23: XIC(S_RCS_EvacSpeedStart_TON.DN)XIO(S_C1_InEvacPosition)OTL(A_C1_0231);
END_ROUTINE
